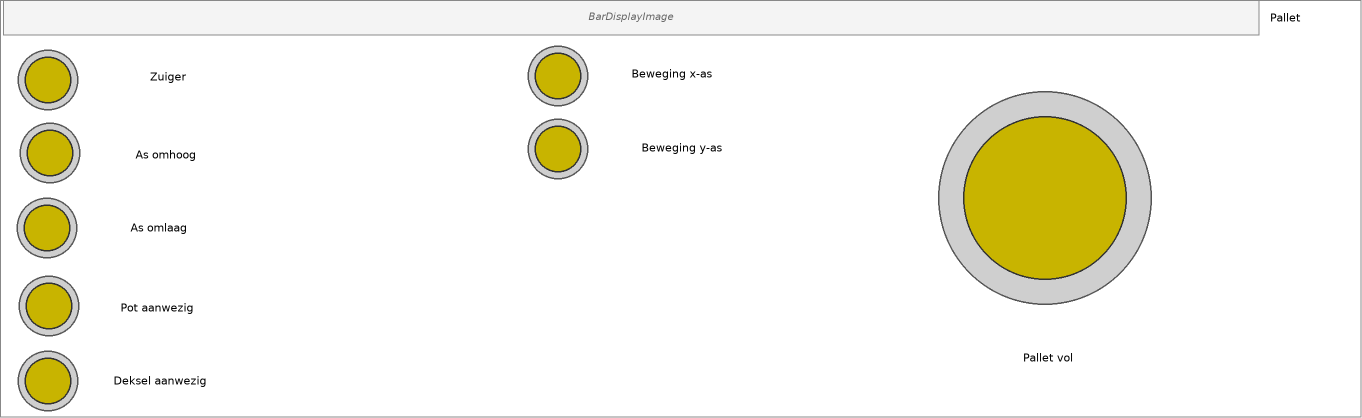
VISUALIZATION Visualization  // 1362x418
    Label (1211,3 149x30), "Pallet"
    Lamp1 (13,45 70x70), variable: GVL_IO.Vplus_Vacuum_start, style: Lamp-Lamp1-Yellow
    Label (93,62 150x30), "Zuiger"
    Lamp1 (15,118 70x70), variable: GVL_IO.a_0_Vertical_Zaxis_upward, style: Lamp-Lamp1-Yellow
    Label (91,140 150x30), "As omhoog"
    Lamp1 (12,193 70x70), variable: GVL_IO.a_1_Vertical_Zaxis_downward, style: Lamp-Lamp1-Yellow
    Label (84,213 150x30), "As omlaag"
    Lamp1 (14,271 70x70), variable: GVL_IO.dp1_Can_detection, style: Lamp-Lamp1-Yellow
    Label (82,293 150x30), "Pot aanwezig"
    Lamp1 (13,346 70x70), variable: GVL_IO.dp2_Cover_detection, style: Lamp-Lamp1-Yellow
    Label (85,366 150x30), "Deksel aanwezig"
    Lamp1 (523,41 70x70), variable: GVL_IO.BUSYX_BUSY_tableX, style: Lamp-Lamp1-Yellow
    Label (597,59 150x30), "Beweging x-as"
    Lamp1 (523,114 70x70), variable: GVL_IO.BUSYY_BUSY_traslationY, style: Lamp-Lamp1-Yellow
    Label (607,133 150x30), "Beweging y-as"
    Lamp1 (921,67 248x262), variable: GVL_IO.BR_Alarm_light, style: Lamp-Lamp1-Yellow
    Label (973,343 150x30), "Pallet vol"
    BarDisplayImage (3,-2 1256x37), value: MAIN.ActualPos, style: BarDisplayImage-Gray, scale format: %.1f, scale 0..25
END_VISUALIZATION

(* stored: Version 1.1.0.1, ProductVersion 3.1.4022.12
   Visu Visualization: Id {215ce958-63df-4c83-b26f-5087e0c38bd6} *)
